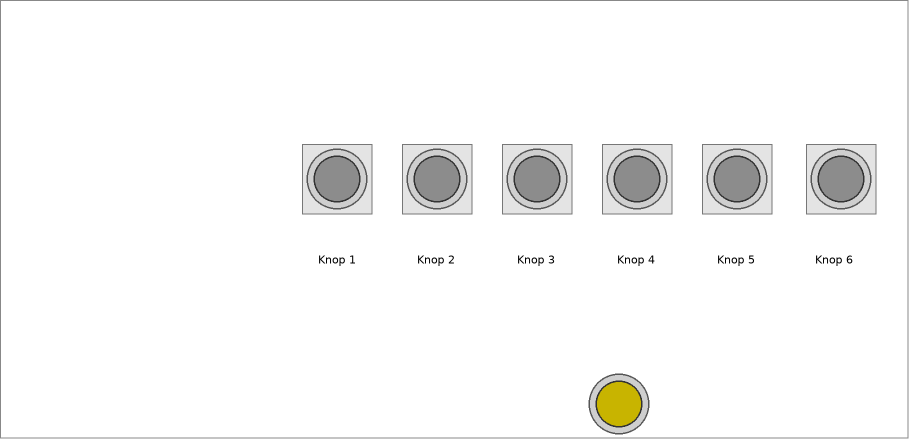
VISUALIZATION Visu  // 909x439
    PushSwitch (302,144 70x70), variable: MAIN.bKnop1, behaviour: TAP, style: Switch-PushSwitch-Gray
    PushSwitch (402,144 70x70), variable: MAIN.bKnop2, behaviour: TAP, style: Switch-PushSwitch-Gray
    PushSwitch (502,144 70x70), variable: MAIN.bKnop3, behaviour: TAP, style: Switch-PushSwitch-Gray
    PushSwitch (602,144 70x70), variable: MAIN.bKnop4, behaviour: TAP, style: Switch-PushSwitch-Gray
    PushSwitch (806,144 70x70), variable: MAIN.bKnop6, behaviour: TAP, style: Switch-PushSwitch-Gray
    PushSwitch (702,144 70x70), variable: MAIN.bKnop5, behaviour: TAP, style: Switch-PushSwitch-Gray
    Label (262,245 150x30), "Knop 1"
    Label (361,245 150x30), "Knop 2"
    Label (461,245 150x30), "Knop 3"
    Label (561,245 150x30), "Knop 4"
    Label (661,245 150x30), "Knop 5"
    Label (759,245 150x30), "Knop 6"
    Lamp1 (584,369 70x70), variable: MAIN.bLamp, style: Lamp-Lamp1-Yellow
END_VISUALIZATION

(* stored: Version 1.1.0.1, ProductVersion 3.1.4024.12
   Visu Visu: Id {d070e602-25e9-49a6-9432-d3b75e6e59d3} *)
